// LS Electric XG5000 project: 9_3
// PLC LSPLC
// module base 0 slot 0: 입출력 모듈:XBC-DR14E (DC 24V 입력 8점, 릴레이 출력 6점)

PROGRAM NewProgram (task: 스캔 프로그램)

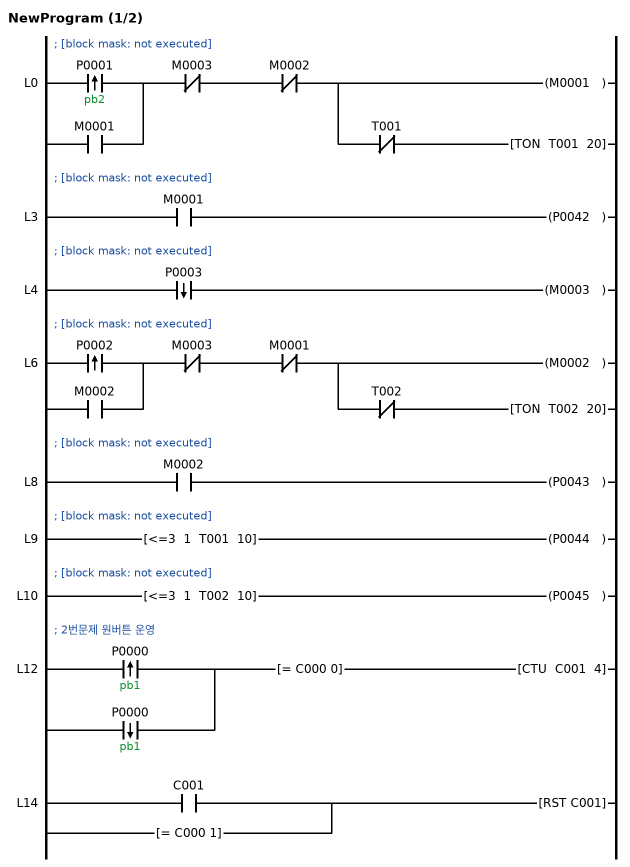
; L0 (block mask: not executed)
LOADP     P0001	// pb2
OR        M0001
AND NOT   M0003
AND NOT   M0002
OUT       M0001
AND NOT   T001
TON       T001 20
; L3 (block mask: not executed)
LOAD      M0001
OUT       P0042
; L4 (block mask: not executed)
LOADN     P0003
OUT       M0003
; L6 (block mask: not executed)
LOADP     P0002
OR        M0002
AND NOT   M0003
AND NOT   M0001
OUT       M0002
AND NOT   T002
TON       T002 20
; L8 (block mask: not executed)
LOAD      M0002
OUT       P0043
; L9 (block mask: not executed)
LOAD<=3   1 T001 10
OUT       P0044
; L10 (block mask: not executed)
LOAD<=3   1 T002 10
OUT       P0045
// 2번문제 원버튼 운영
; L12
LOADP     P0000	// pb1
ORN       P0000	// pb1
AND=      C000 0
CTU       C001 4
; L14
LOAD      C001
OR=       C000 1
RST       C001

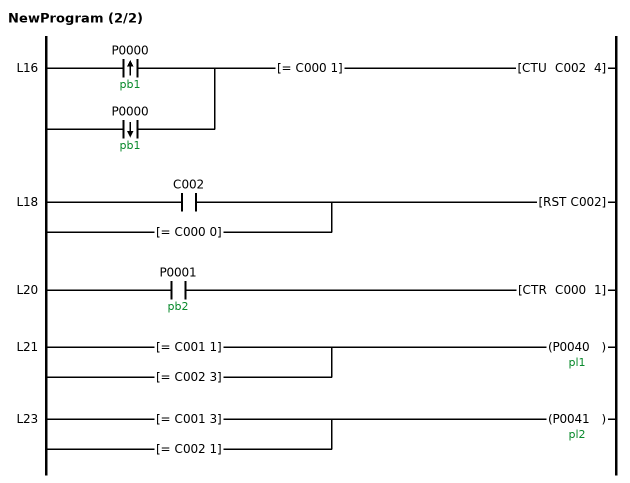
; L16
LOADP     P0000	// pb1
ORN       P0000	// pb1
AND=      C000 1
CTU       C002 4
; L18
LOAD      C002
OR=       C000 0
RST       C002
; L20
LOAD      P0001	// pb2
CTR       C000 1
; L21
LOAD=     C001 1
OR=       C002 3
OUT       P0040	// pl1
; L23
LOAD=     C001 3
OR=       C002 1
OUT       P0041	// pl2